FUNCTION_BLOCK viritual_control_box //IMPLEMENTS if_controller
VAR_INPUT
END_VAR
VAR_OUTPUT
END_VAR
VAR
END_VAR

METHOD joystick : REAL
VAR_INPUT
END_VAR
END_METHOD

METHOD mode : enum_switch
VAR_INPUT
END_VAR
END_METHOD

METHOD status : sys_stat
VAR_INPUT
END_VAR
VAR_OUTPUT
	current_sys_stat : sys_stat;
END_VAR
VAR
	have_start_been_high : BOOL := FALSE;
	have_stop_been_high : BOOL := FALSE;
END_VAR
IF GVL.start_Button = TRUE THEN
	current_sys_stat := sys_stat.ready;
ELSIF GVL.start_Button = FALSE THEN
	current_sys_stat := sys_stat.fault;
ELSE
	current_sys_stat := sys_stat.notReady;
END_IF
END_METHOD

END_FUNCTION_BLOCK

(* stored: Version 1.1.0.1, ProductVersion 3.1.4024.12
   POU viritual_control_box: Id {906cb42c-d2ed-4599-9ef1-b92485558ae5}, SpecialFunc None
   Method joystick: Id {14014bdd-18c6-4c0e-89e5-910e597357d8}
   Method mode: Id {4a202379-5761-4478-9728-4c281ca12f57}
   Method status: Id {90598556-d513-4ee8-9db4-63caba628b1e} *)
